// ---- Machine/VISUs/V_Main.TcVIS
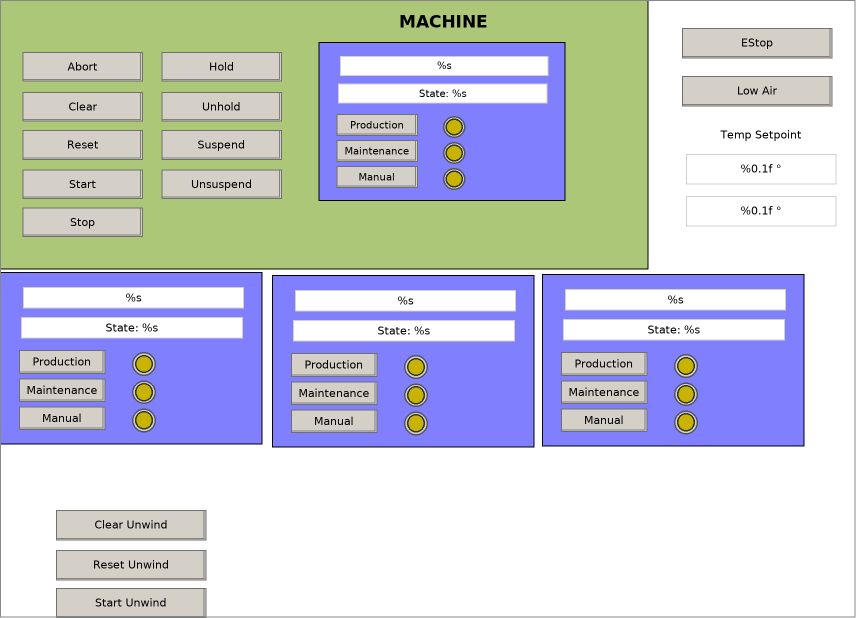
VISUALIZATION V_Main  // 856x618
    Frame (0,0 856x269)
        shows V_MachineModule(HMI := MAIN.VFFSDemo.PackMLBaseModule_HMI)
    Frame (0,272 262x172)
        shows V_Module(HMI := MAIN.VFFSDemo.PullWheels.PackMLBaseModule_HMI)
    Frame (272,275 262x172)
        shows V_Module(HMI := MAIN.VFFSDemo.Sealer.PackMLBaseModule_HMI)
    Frame (542,274 262x172)
        shows V_Module(HMI := MAIN.VFFSDemo.Unwind.PackMLBaseModule_HMI)
    Button (682,28 150x30), "EStop"
        toggle MAIN.VFFSDemo.EstopInput
    Button (682,76 150x30), "Low Air"
        toggle MAIN.VFFSDemo.LowAirInput
    Textfield (686,154 150x30), "%0.1f °", text variable: MAIN.VFFSDemo.Sealer.SealBar._SetTemperature
        OnMouseDown: write the text variable via VisuDialogs.Numpad, min 20, max 400, title 'Sealer Bar Temp Setpoint', format %0.1f
    Label (686,120 150x30), "Temp Setpoint"
    Textfield (686,196 150x30), "%0.1f °", text variable: MAIN.VFFSDemo.Sealer.SealBar._ActualTemperature
    Button (56,510 150x30), "Clear Unwind"
        OnMouseClick: execute { MAIN.VFFSDemo.unwind.PackMLBaseModule_HMI.Command.State := E_PMLCommand.ePMLCommand_Clear; }
    Button (56,550 150x30), "Reset Unwind"
        OnMouseClick: execute { MAIN.VFFSDemo.unwind.PackMLBaseModule_HMI.Command.State := E_PMLCommand.ePMLCommand_Reset; }
    Button (56,588 150x30), "Start Unwind"
        OnMouseClick: execute { MAIN.VFFSDemo.unwind.PackMLBaseModule_HMI.Command.State := E_PMLCommand.ePMLCommand_Start; }
END_VISUALIZATION
